# EPICS alarm handler configuration: alh_files/mgnt_ltu_kick.alhConfig
GROUP NULL KICK:LTU1:MG01
   $COMMAND edm -x -eolc -noedit mgnt_ltu1_kick.edl
$ALIAS KICK
$GUIDANCE
LTU1 KICK
   Group Name: KICK:LTU1:MG01
   Summary PV:  KICK:LTU1:MG01:STATSUMY
$END

GROUP KICK:LTU1:MG01  KICK:LTU1:320
   $COMMAND edm -x -eolc -noedit -m "DEV=KICK:LTU1:320" mgnt_unit.edl
CHANNEL    KICK:LTU1:320    KICK:LTU1:320:STATMSG   -----
   $FORCEPV KICK:LTU1:320:STATMSGSV -DATL 1 0
